// TIA Portal project "PLCII_Pro6" (V15.1)

(* hardware
DEVICE "S7-1200 station_1"  S7-1200 Station
   slot 0: "Rack_0"  S7-1200 Rack  Rack  V1.0
   slot 1: "PLC_1"  CPU 1215C DC/DC/Rly  6ES7 215-1HG40-0XB0  V4.2
*)

// ===== PLC "PLC_1"  CPU 1215C DC/DC/Rly =====

VAR_GLOBAL   // PLC tag table "Default tag table"
   "Start" AT %M0.0 : Bool;
   "Sys_runing" AT %M0.1 : Bool;
   "Stop" AT %M0.2 : Bool;
   "Activate" AT %M0.3 : Bool;
   "Sys_Activated" AT %M0.4 : Bool;
END_VAR

DATA_BLOCK "SysVaribales"   // DB1
{ S7_Optimized_Access := 'TRUE' }
VERSION : 0.1
   VAR
      Seconds : Time;
      Minutes : Int;
      Hours : Int;
      Hours1000 : Int;
      Reset : Bool;
      FirstIND : Time;
   END_VAR
BEGIN
END_DATA_BLOCK

DATA_BLOCK "Hourmeter_DB"   // DB2
{ S7_Optimized_Access := 'TRUE' }
VERSION : 0.1
// stored: InstanceOfName Hourmeter
"Hourmeter"
BEGIN
END_DATA_BLOCK

// folder: System blocks/Program resources

DATA_BLOCK "IEC_Timer_0_DB"   // DB3
{ S7_Optimized_Access := 'TRUE' }
AUTHOR : Simatic
FAMILY : IEC
NAME : IEC_TMR
VERSION : 1.0
// stored: InstanceOfName IEC_TIMER
"IEC_TIMER"
BEGIN
END_DATA_BLOCK

// folder: (top level)

FUNCTION_BLOCK "Hourmeter"   // FB1, LAD
{ S7_Optimized_Access := 'TRUE' }
VERSION : 0.1
   VAR RETAIN
      Counter1 : IEC_COUNTER;
      Counter2 : IEC_COUNTER;
      ons1 : Bool;
   END_VAR
   VAR
      ons2 : Bool;
      ons3 : Bool;
      ons4 : Bool;
      ons5 : Bool;
      ons6 : Bool;
      ons7 : Bool;
      ons8 : Bool;
      ons9 : Bool;
      ons10 : Bool;
      ResetC1 : Bool;
      ResetC2 : Bool;
      ResResetC1 : Bool;
      ResResetC2 : Bool;
      oki : Bool;
   END_VAR
   VAR_TEMP
      SecTEMP : Time;
   END_VAR
   VAR_TEMP   // added for the SCL form of the ladder/FBD networks
      _w1 : Bool;
      _w2 : Bool;
   END_VAR
BEGIN

REGION Network 1
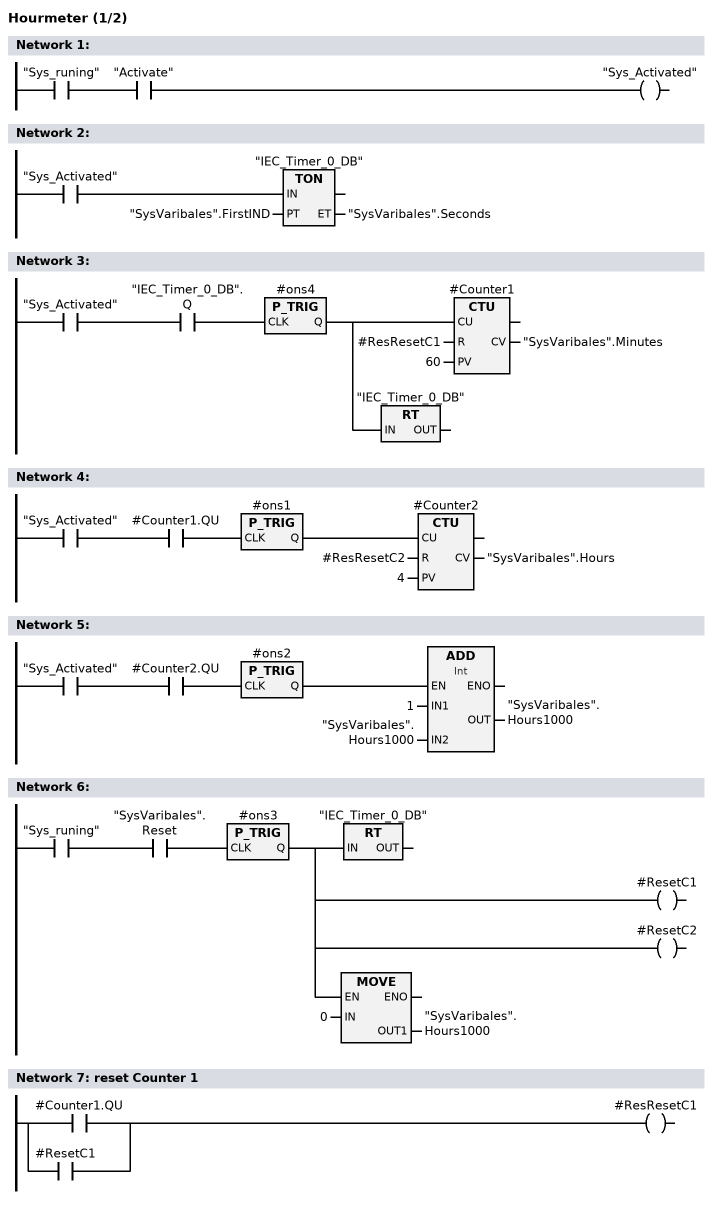
   RUNG wire#powerrail
      Contact( "Sys_runing" )
      Contact( "Activate" )
      Coil( "Sys_Activated" )
   END_RUNG
   // the same network as SCL:
   "Sys_Activated" := "Sys_runing" AND "Activate";
END_REGION

REGION Network 2
   "IEC_Timer_0_DB".TON(IN := "Sys_Activated", PT := "SysVaribales".FirstIND, ET => "SysVaribales".Seconds);
END_REGION

REGION Network 3
   #_w1 := "Sys_Activated" AND "IEC_Timer_0_DB".Q;
   #_w2 := #_w1 AND NOT #ons4;   // rising edge
   #ons4 := #_w1;
   #Counter1.CTU(CU := #_w2, R := #ResResetC1, PV := 60, CV => "SysVaribales".Minutes);
   IF #_w2 THEN RESET_TIMER("IEC_Timer_0_DB"); END_IF;
END_REGION

REGION Network 4
   #_w1 := "Sys_Activated" AND #Counter1.QU;
   #_w2 := #_w1 AND NOT #ons1;   // rising edge
   #ons1 := #_w1;
   #Counter2.CTU(CU := #_w2, R := #ResResetC2, PV := 4, CV => "SysVaribales".Hours);
END_REGION

REGION Network 5
   RUNG wire#powerrail
      Contact( "Sys_Activated" )
      Contact( #Counter2.QU )
      P_Trig( #ons2 )
      { S7_Templates := "SrcType := Int" } Add(in1 := 1, in2 := "SysVaribales".Hours1000, out => "SysVaribales".Hours1000)
   END_RUNG
   // the same network as SCL:
   #_w1 := "Sys_Activated" AND #Counter2.QU;
   #_w2 := #_w1 AND NOT #ons2;   // rising edge
   #ons2 := #_w1;
   IF #_w2 THEN "SysVaribales".Hours1000 := 1 + "SysVaribales".Hours1000; END_IF;
END_REGION

REGION Network 6
   RUNG wire#powerrail
      Contact( "Sys_runing" )
      Contact( "SysVaribales".Reset )
      P_Trig( #ons3 )
      wire#w1
      RT_Coil( "IEC_Timer_0_DB" )
   END_RUNG
   RUNG wire#w1
      Coil( #ResetC1 )
   END_RUNG
   RUNG wire#w1
      Coil( #ResetC2 )
   END_RUNG
   RUNG wire#w1
      Move(in := 0, out1 => "SysVaribales".Hours1000)
   END_RUNG
   // the same network as SCL:
   #_w1 := "Sys_runing" AND "SysVaribales".Reset;
   #_w2 := #_w1 AND NOT #ons3;   // rising edge
   #ons3 := #_w1;
   IF #_w2 THEN RESET_TIMER("IEC_Timer_0_DB"); END_IF;
   #ResetC1 := #_w2;
   #ResetC2 := #_w2;
   IF #_w2 THEN "SysVaribales".Hours1000 := 0; END_IF;
END_REGION

REGION Network 7: reset Counter 1
   RUNG wire#powerrail
      Contact( #Counter1.QU )
      wire#w1
      Coil( #ResResetC1 )
   END_RUNG
   RUNG wire#powerrail
      Contact( #ResetC1 )
   END_RUNG wire#w1
   // the same network as SCL:
   #ResResetC1 := #Counter1.QU OR #ResetC1;
END_REGION

REGION Network 8: reset Counter 1
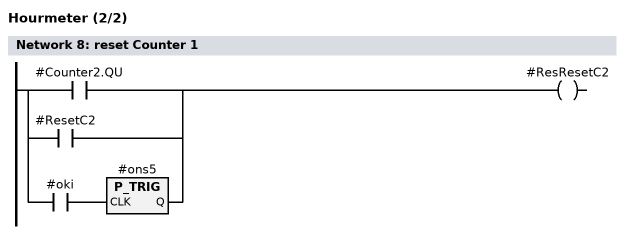
   RUNG wire#powerrail
      Contact( #Counter2.QU )
      wire#w1
      Coil( #ResResetC2 )
   END_RUNG
   RUNG wire#powerrail
      Contact( #ResetC2 )
   END_RUNG wire#w1
   RUNG wire#powerrail
      Contact( #oki )
      P_Trig( #ons5 )
   END_RUNG wire#w1
   // the same network as SCL:
   #_w1 := #oki AND NOT #ons5;   // rising edge
   #ons5 := #oki;
   #ResResetC2 := #Counter2.QU OR #ResetC2 OR #_w1;
END_REGION
END_FUNCTION_BLOCK

ORGANIZATION_BLOCK "Main"   // OB1, LAD, ProgramCycle
TITLE = "Main Program Sweep (Cycle)"
{ S7_Optimized_Access := 'TRUE' }
VERSION : 0.1
   VAR_INPUT
      Initial_Call : Bool;   // Initial call of this OB
      Remanence : Bool;   // =True, if remanent data are available
   END_VAR
BEGIN

REGION Network 1
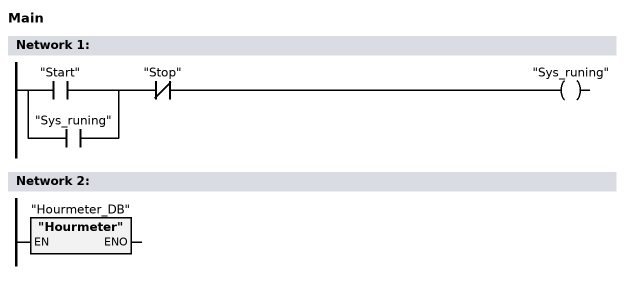
   RUNG wire#powerrail
      Contact( "Start" )
      wire#w1
      I_Contact( "Stop" )
      Coil( "Sys_runing" )
   END_RUNG
   RUNG wire#powerrail
      Contact( "Sys_runing" )
   END_RUNG wire#w1
   // the same network as SCL:
   "Sys_runing" := ("Start" OR "Sys_runing") AND NOT "Stop";
END_REGION

REGION Network 2
   RUNG wire#powerrail
      "Hourmeter_DB"()
   END_RUNG
   // the same network as SCL:
   "Hourmeter_DB"();   // "Hourmeter"
END_REGION
END_ORGANIZATION_BLOCK